PROGRAM MAIN

DevicesExample();
ForceableExample();
DevicesPolymorphismExample();
GVL_Forceables.manager.renew();

END_PROGRAM

(* stored: Version 1.1.0.1, ProductVersion 3.1.4026.18
   POU MAIN: Id {1593e7da-0106-4d2c-9dea-9594914e3509}, SpecialFunc None *)
